(* PLC project Unbenannt, Unbekannt Unbenannt 1 *)
(* stored: creationDateTime 2019-05-29T14:07:24, modificationDateTime 2019-08-11T20:04:34 *)

FUNCTION_BLOCK PT_Calc
  VAR_INPUT
    Rtd : REAL;  (* Value from MAX Chip *)
    R_0_Grad : REAL;  (* Resistance at 0° C; PT100=100R; PT1000=1000R *)
  END_VAR
  VAR
    R_0_Norm : REAL;  (* Normalized to 100R; Enables to use PT100 und PT1000 *)
  END_VAR
  VAR_INPUT
    R_Ref : REAL;  (* Referance resistor; PT100=430R; PT1000=4300R *)
  END_VAR
  VAR_OUTPUT
    Ratio : REAL;
    R_Ist : REAL;  (* actual resistance *)
  END_VAR
  VAR CONSTANT
    K_32768 : REAL := 32768.0;
    a : REAL := 3.9083E-03;
    b : REAL := -5.7750E-07;
    c : REAL := -4.1830E-12;
    K_2 : REAL := 2.0;
    K_3 : REAL := 3.0;
    K_4 : REAL := 4.0;
    K_5 : REAL := 5.0;
    K_100 : REAL := 100.0;
    K_min1 : REAL := -1.0;
  END_VAR
  VAR_OUTPUT
    Temp : REAL;
  END_VAR
  VAR CONSTANT
    K_a_kl0 : REAL := 2.2228;  (* Temp < 0°C *)
    K_b_kl0 : REAL := 2.5859E-3;  (* Temp < 0°C *)
    K_c_kl0 : REAL := 4.8260E-6;  (* Temp < 0°C *)
    K_d_kl0 : REAL := 2.8183E-8;  (* Temp < 0°C *)
    K_e_kl0 : REAL := 1.5243E-10;  (* Temp < 0°C *)
    K_242_02 : REAL := 242.02;  (* Temp < 0°C *)
  END_VAR
  VAR  (* added by the conversion: wires and edge detectors of the diagram *)
    _GE78_OUT : BOOL;
  END_VAR

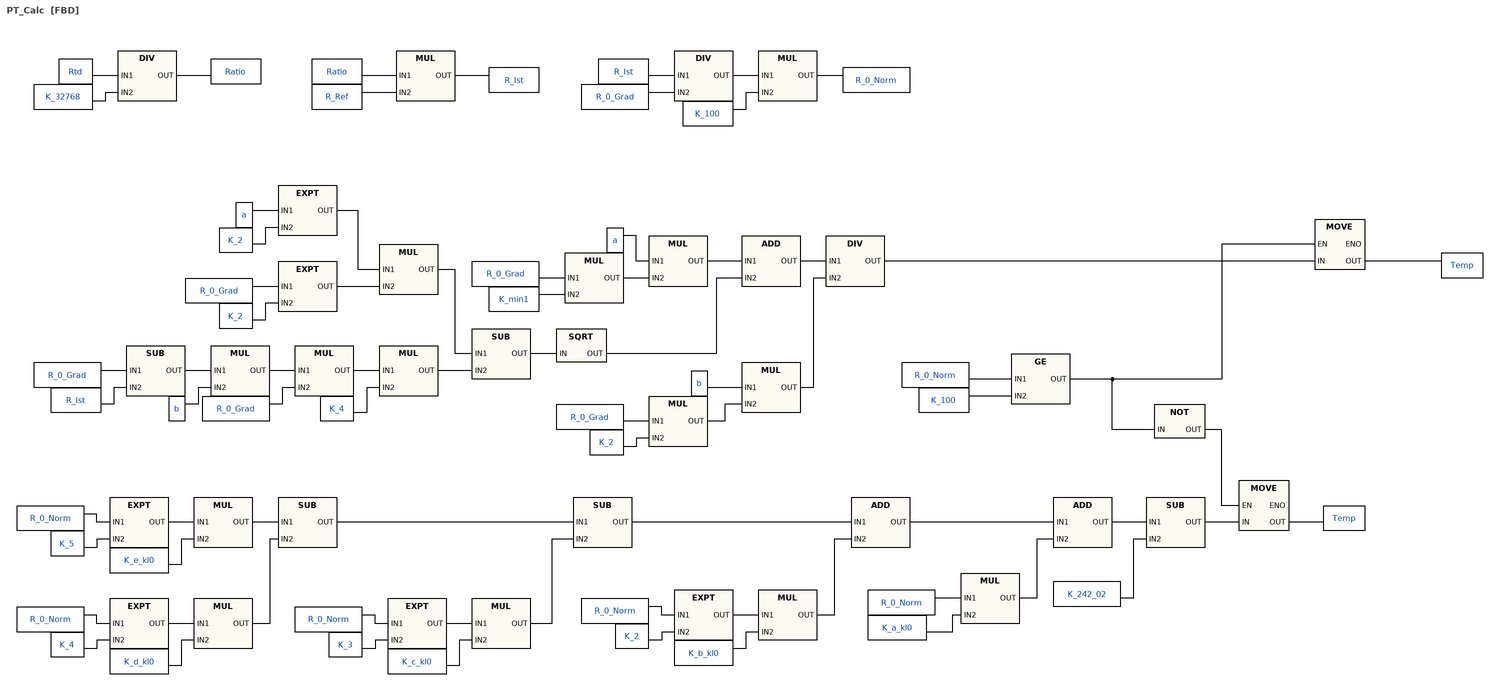
(* FBD diagram, written out as Structured Text *)
Ratio := Rtd / K_32768;
R_Ist := Ratio * R_Ref;
R_0_Norm := R_Ist / R_0_Grad * K_100;
_GE78_OUT := R_0_Norm >= K_100;
IF _GE78_OUT THEN Temp := (a * (R_0_Grad * K_min1) + SQRT(EXPT(a, K_2) * EXPT(R_0_Grad, K_2) - (R_0_Grad - R_Ist) * b * R_0_Grad * K_4)) / (b * (R_0_Grad * K_2)); END_IF;
IF NOT _GE78_OUT THEN Temp := EXPT(R_0_Norm, K_5) * K_e_kl0 - EXPT(R_0_Norm, K_4) * K_d_kl0 - EXPT(R_0_Norm, K_3) * K_c_kl0 + EXPT(R_0_Norm, K_2) * K_b_kl0 + R_0_Norm * K_a_kl0 - K_242_02; END_IF;
END_FUNCTION_BLOCK

FUNCTION_BLOCK Well_pak_steu
  VAR
    TP0 : TP;
    RS0 : RS;
    F_TRIG0 : F_TRIG;
    F_TRIG1 : F_TRIG;
    Summe : INT;
    K_100 : INT := 100;
  END_VAR
  VAR_OUTPUT
    SSR : BOOL;  (* zero crossing ssr needed *)
  END_VAR
  VAR_INPUT
    Start : BOOL := False;
  END_VAR
  VAR
    K_T_02 : TIME := T#20ms;
  END_VAR
  VAR_INPUT
    Percent_Power : INT := 0;
  END_VAR
  VAR  (* added by the conversion: wires and edge detectors of the diagram *)
    _GE8_OUT : BOOL;
    _ADD35_ENO : BOOL;
    _ADD35_OUT : INT;
  END_VAR

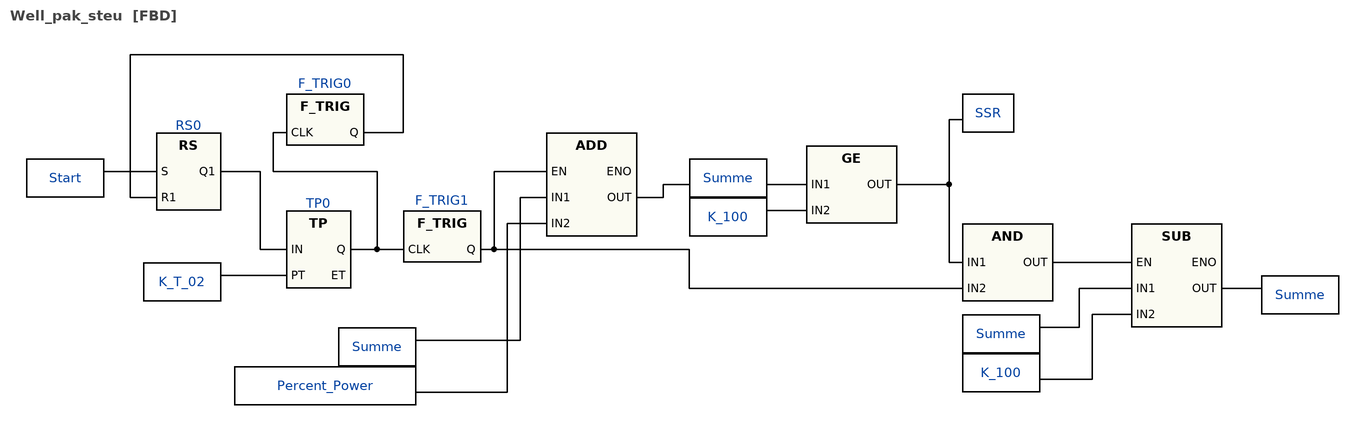
(* FBD diagram, written out as Structured Text *)
_GE8_OUT := Summe >= K_100;
SSR := _GE8_OUT;
F_TRIG0(CLK := TP0.Q);
RS0(S := Start, R1 := F_TRIG0.Q);
TP0(IN := RS0.Q1, PT := K_T_02);
F_TRIG1(CLK := TP0.Q);
_ADD35_OUT := ADD(EN := F_TRIG1.Q, IN1 := Summe, IN2 := Percent_Power, ENO => _ADD35_ENO);
IF _ADD35_ENO THEN Summe := _ADD35_OUT; END_IF;
IF _GE8_OUT AND F_TRIG1.Q THEN Summe := Summe - K_100; END_IF;
END_FUNCTION_BLOCK

(* Schaltet aus bei IN < Low; Schaltet ein bei IN > High *)
FUNCTION_BLOCK Hysterese2
  VAR_INPUT
    IN : WORD;
    Low : WORD;
    High : WORD;
  END_VAR
  VAR_OUTPUT
    Out : BOOL;
  END_VAR

            IF in < low THEN
	Out := FALSE;
ELSIF in > high THEN
	Out := TRUE;
END_IF;




(* revision history
hm		4.  aug. 2006	rev 1.0
	original version

hm		2. jun. 2008	rev 1.1
	improved performance
*)
          
END_FUNCTION_BLOCK

PROGRAM program0
  VAR
    Hysterese20 : Hysterese2;
  END_VAR

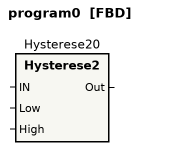
(* FBD diagram, written out as Structured Text *)
Hysterese20();
END_PROGRAM

FUNCTION_BLOCK Two_Steps_Burner_PID
  VAR_INPUT
    Start : BOOL;
    T_Set : REAL;
    T_act : REAL;
  END_VAR
  VAR
    XO : REAL := 0.0;  (* Ausgangswert bei Auto = False *)
    KP : REAL;
    TR : REAL;
    TD : REAL;
    Cycle : TIME := T#1s;
  END_VAR
  VAR_OUTPUT
    Burner_on : BOOL;
    Level_1 : BOOL;
    Level_2 : BOOL;
  END_VAR
  VAR
    PID0 : PID;
    L_Min : WORD := 0;  (* lower border PID out *)
    L_Max : WORD := 1000;  (* upper border PID out *)
    Hysterese20 : Hysterese2;
    Hysterese21 : Hysterese2;
    Low_ST1 : WORD := 450;
    High_ST1 : WORD := 500;
    Low_ST2 : WORD := 650;
    High_ST2 : WORD := 700;
  END_VAR
  VAR  (* added by the conversion: wires and edge detectors of the diagram *)
    _LIMIT10_OUT : WORD;
  END_VAR

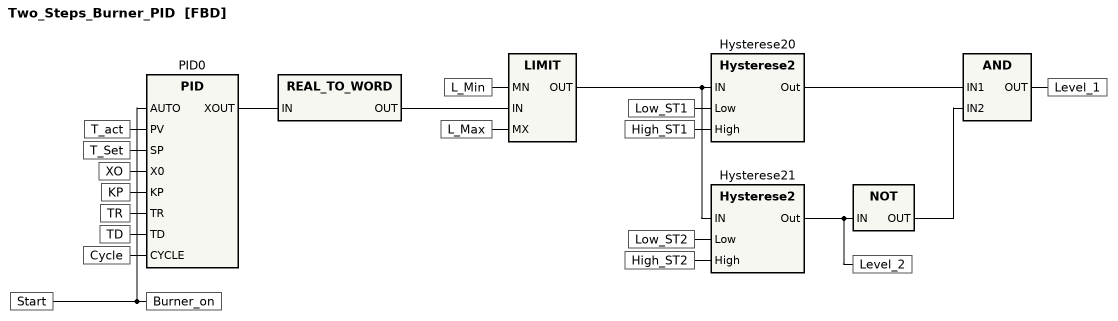
(* FBD diagram, written out as Structured Text *)
Burner_on := Start;
PID0(AUTO := Start, PV := T_act, SP := T_Set, X0 := XO, KP := KP, TR := TR, TD := TD, CYCLE := Cycle);
_LIMIT10_OUT := LIMIT(L_Min, REAL_TO_WORD(PID0.XOUT), L_Max);
Hysterese20(IN := _LIMIT10_OUT, Low := Low_ST1, High := High_ST1);
Hysterese21(IN := _LIMIT10_OUT, Low := Low_ST2, High := High_ST2);
Level_1 := Hysterese20.Out AND NOT Hysterese21.Out;
Level_2 := Hysterese21.Out;
END_FUNCTION_BLOCK

(* Eingabe Analoger Wert (0-1023) Ausgabe Reale Temperatur *)
FUNCTION_BLOCK Analog_IN_Realtemp_OUT
  VAR
    Res_IN : WORD := 1023;  (* Resolution of Input i.e.: 0-1023 = 1024 *)
    PT_Range : WORD := 150;  (* Range of transmitter; i.e. 0-150°C = 150 *)
  END_VAR
  VAR_INPUT
    MW_act : WORD;  (* actual value *)
  END_VAR
  VAR_OUTPUT
    MW_Ist0 : REAL;  (* Temperature in °C *)
  END_VAR

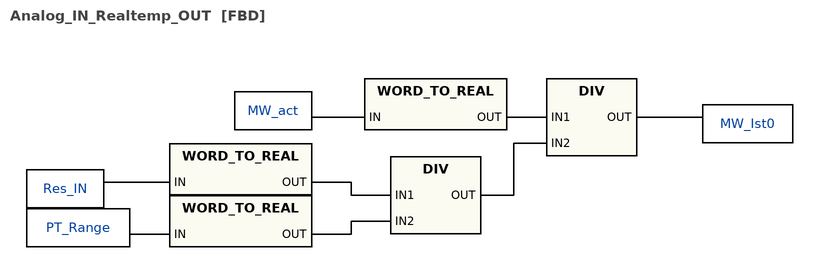
(* FBD diagram, written out as Structured Text *)
MW_Ist0 := WORD_TO_REAL(MW_act) / (WORD_TO_REAL(Res_IN) / WORD_TO_REAL(PT_Range));
END_FUNCTION_BLOCK

FUNCTION_BLOCK Rnd_any_DecPt
  VAR_INPUT
    IN_Real : REAL;
  END_VAR
  VAR_OUTPUT
    Out_Real_rounded : REAL;
  END_VAR
  VAR_INPUT
    Dec_Pt : INT;
  END_VAR
  VAR  (* added by the conversion: wires and edge detectors of the diagram *)
    _EXP3_OUT : REAL;
  END_VAR

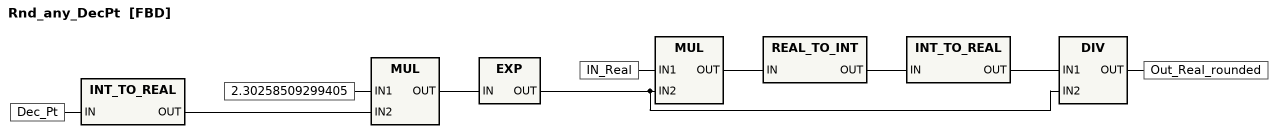
(* FBD diagram, written out as Structured Text *)
_EXP3_OUT := EXP(2.30258509299405 * INT_TO_REAL(Dec_Pt));
Out_Real_rounded := INT_TO_REAL(REAL_TO_INT(IN_Real * _EXP3_OUT)) / _EXP3_OUT;
END_FUNCTION_BLOCK

CONFIGURATION Config0
  RESOURCE Res0 ON PLC
    TASK task0(INTERVAL := T#20ms, PRIORITY := 0);
    PROGRAM instance0 WITH task0 : program0;
  END_RESOURCE
END_CONFIGURATION
